Staubli VAL3: RosSimpleMsg.dtx

mdesc mNomSpeed
public Header header
  [0]
    num nMsgType
    num nCommType
    num nReplyCode
public Prefix prefix
  [0]
    num nLength
public Body body
  [0]
    num nData
